FUNCTION_BLOCK FB_PCMSupplySystem EXTENDS FB_SystemContinous
VAR_INPUT
	nControlModeAutomatic : E_PCMSystemControlMode;
	
END_VAR
VAR_OUTPUT
END_VAR
VAR
	
	{attribute 'OPC.UA.DA' := '1'}
	localSetParameters : ST_PCMSystemSetParameters;
	
	//heat meters
	WMZ900 : FB_MollineUltramess403HeatCounter; //pcm storage
	WMZ935 : FB_MollineUltramess403HeatCounter; //chiller
	
	//temperature sensors
	
	TS901 : FB_TemperatureSensor_KL3214;
	TS902 : FB_TemperatureSensor_KL3214;
	TS903 : FB_TemperatureSensor_KL3214;
	TS910 : FB_TemperatureSensor_KL3214;
	TS911 : FB_TemperatureSensor_KL3214;
	TS950 : FB_TemperatureSensor_KL3214;
	TS951 : FB_TemperatureSensor_KL3214;
	
	//valves
	ST_RV950DefaultParameters : ST_MixingValveDefaultParameters := (bFeedbackSignal := FALSE, tTaskCycleTime := GlobalVariables.tTaskCycleTime_MAIN, tCtrlCycleTime := GlobalVariables.tCtrlCycleTime_MAIN);
	RV950 : FB_MixingValve := (ST_DefaultParameters := ST_RV950DefaultParameters);
	
	// pcm chiller
	PCMChiller : FB_PCMChiller;
	
	// PCMStorage
	PCMStorage : FB_PCMStorage;
	
	//internal variables
	nControlMode : E_PCMSystemControlMode;
	
	bSetStatusOn_RV950 : BOOL; 
	
	
END_VAR

SelectLocalControlMode();


WMZ900(aHeatCounterTelegramm := aTelegramm_WMZ900);
WMZ935(aHeatCounterTelegramm := aTelegramm_WMZ935);
	
TS901();
TS901.GetState_AI();
TS902();
TS902.GetState_AI();
TS903();
TS903.GetState_AI();
TS910();
TS910.GetState_AI();
TS911();
TS911.GetState_AI();
TS950();
TS950.GetState_AI();
TS951();
TS951.GetState_AI();

RV950.GetState_AI();
RV950(bSetStatusOnAutomatic := bSetStatusOn_RV950,
	fSetPointAutomatic := 100,
	bAlgorithmPermission := TRUE,
	fTemperatureExternal := TS950.fTemperature,
	nControlModeAutomatic := 0);
RV950.SetState_AO();

PCMChiller.GetState(); 
PCMChiller(bSetStatusOnAutomatic := FALSE, 
	bAlgorithmPermission := bAlgorithmPermission,
	fSetPointAutomatic := fSetPoint);
PCMChiller.SetState();

METHOD PROTECTED  CheckError : BOOL
VAR_INPUT
END_VAR
VAR_OUTPUT
	bError : BOOL;
END_VAR
END_METHOD

METHOD LocalControl : BOOL
VAR_INPUT
	
END_VAR
CASE nControlMode OF
	0: //stand-by
	PCMChiller.bStatusOn := FALSE; 
	 	
	1: //direct cooling 
	PCMChiller.nControlModeAutomatic := 0; 
	PCMChiller.fSetPointAutomatic := fSetPoint; 
	bSetStatusOn_RV950 := FALSE; 
	
	2: //charge pcm
	PCMChiller.nControlModeAutomatic := 0; 
	PCMChiller.fSetPointAutomatic := fSetPoint;
	bSetStatusOn_RV950 := TRUE; 
	
	3: //discharge pcm
	PCMChiller.nControlModeAutomatic := 1; 
	bSetStatusOn_RV950 := TRUE; 
		
END_CASE
END_METHOD

METHOD PROTECTED  Operational : BOOL
VAR_INPUT
END_VAR
VAR_OUTPUT
	bSwitchToWorking : BOOL := FALSE;
END_VAR
END_METHOD

METHOD PROTECTED  RampDown : BOOL
VAR_INPUT
END_VAR
VAR_OUTPUT
	bRampDownFinished : BOOL := FALSE;
END_VAR
END_METHOD

METHOD PROTECTED  RampUp : BOOL
VAR_INPUT
END_VAR
VAR_OUTPUT
	bRampUpFinished : BOOL := TRUE;
END_VAR
END_METHOD

METHOD SelectLocalControlMode : BOOL
VAR_INPUT
END_VAR
IF control.bManualModeActivated THEN
	nControlMode := localSetParameters.nControlModeManual;
ELSIF control.bAlgorithmModeActivated AND bAlgorithmPermission THEN
	nControlMode := localSetParameters.nControlModeAlgorithm;
ELSE
	nControlMode := nControlModeAutomatic;
END_IF
END_METHOD

METHOD PROTECTED   SetSetPointLimits : BOOL
VAR_INPUT
END_VAR
END_METHOD

METHOD PROTECTED  SetState : BOOL
VAR_INPUT
END_VAR
VAR_OUTPUT
END_VAR
END_METHOD

METHOD PROTECTED  Working : BOOL
VAR_INPUT
END_VAR
VAR_OUTPUT
	bSwitchToOperational : BOOL := FALSE;
END_VAR
//Implementing different control modes (next time)
END_METHOD

END_FUNCTION_BLOCK

(* stored: Version 1.1.0.1, ProductVersion 3.1.4024.10
   POU FB_PCMSupplySystem: Id {341025c6-61f6-42b1-9c8c-58df0f661ef4}, SpecialFunc None
   Method CheckError: Id {8839b696-1d9b-4a95-9794-1c9ab39cf8a3}
   Method LocalControl: Id {97954005-d85c-4ab5-8282-6a3311969e99}
   Method Operational: Id {aa3415d6-b9e3-41e4-8cd7-e25495beab13}
   Method RampDown: Id {57928382-ae9d-4c1d-8eb0-92bff3c44af7}
   Method RampUp: Id {91f83af4-cae3-4c39-8ad3-f335a1458b58}
   Method SelectLocalControlMode: Id {9e12ff0b-91fd-4673-8be9-ddb0be52ac97}
   Method SetSetPointLimits: Id {f3c99afb-2328-4e69-8097-2f00253230f8}
   Method SetState: Id {a8999fa2-3070-4e35-8eaa-105279b0b728}
   Method Working: Id {27f0d096-76fc-4f63-bb50-defbb605afdf} *)
